SUBAPPLICATION Uebung_004a3 (* wie Uebung_004a2 aber ohne E_MERGE *)
  (* Standard: 61499-2 *)
  (* Version 1.0, 2023-10-23, franz *)
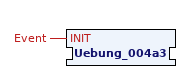
  EVENT_INPUT
    INIT;
  END_EVENT
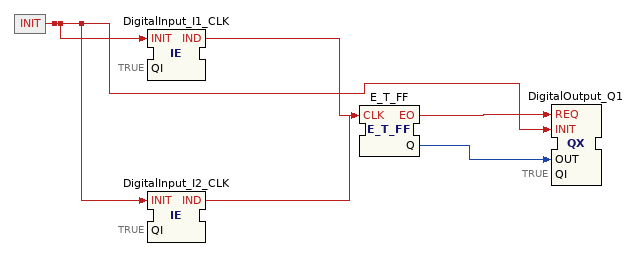
  FBS
    DigitalOutput_Q1 : QX(QI := TRUE);
    DigitalInput_I1_CLK : IE(QI := TRUE);
    E_T_FF : E_T_FF;
    DigitalInput_I2_CLK : IE(QI := TRUE);
  END_FBS
  EVENT_CONNECTIONS
    INIT TO DigitalInput_I1_CLK.INIT;
    E_T_FF.EO TO DigitalOutput_Q1.REQ;
    INIT TO DigitalOutput_Q1.INIT;
    INIT TO DigitalInput_I2_CLK.INIT;
    DigitalInput_I1_CLK.IND TO E_T_FF.CLK;
    DigitalInput_I2_CLK.IND TO E_T_FF.CLK;
  END_CONNECTIONS
  DATA_CONNECTIONS
    E_T_FF.Q TO DigitalOutput_Q1.OUT;
  END_CONNECTIONS
END_SUBAPPLICATION
